(* IEC 61131-3 sources: ai-building-automation/docs/phase0/s3_evidence/dev2/types/generated, 3 files *)

(* ---- PLC_PRG.st ---- *)
PROGRAM PLC_PRG
VAR
    (* Deterministic demo for AHU-01 *)
    StartCommand : BOOL := FALSE;
    StopCommand : BOOL := FALSE;
    FanCommand : BOOL := FALSE;
    FanRunning : BOOL := FALSE;
    FanFault : BOOL := FALSE;
    SupplyTemp : REAL := 21.0;
    Setpoint : REAL := 22.0;
    FanSpeed : REAL := 50.0;
    HeatingValve : REAL := 0.0;
    TestCoil : BOOL := FALSE;
    TestDiscreteInput : BOOL := TRUE;
    TestWordRead : WORD := 16#A55A;
    TestWordWrite : WORD := 16#0000;
    TestInt16Read : INT := -1234;
    TestInt16Write : INT := 0;
    TestUInt16Read : UINT := 1234;
    TestUInt16Write : UINT := 0;
    TestReal32Read : REAL := 21.5;
    TestReal32Write : REAL := 0.0;
    (* Modbus TCP image (16-bit words, mapped to Modbus_TCP_Server I/O) *)
    Mb_Command : WORD; (* HR0 Command: bit0=StartCommand, bit1=StopCommand *)
    Mb_TestInt16Write : WORD; (* HR1 TestInt16Write INT16 WRITE *)
    Mb_TestReal32Write_W0 : WORD; (* HR2 TestReal32Write REAL32 memory word 0 *)
    Mb_TestReal32Write_W1 : WORD; (* HR3 TestReal32Write REAL32 memory word 1 *)
    p_TestReal32Write : POINTER TO ARRAY[0..1] OF WORD;
    Mb_TestUInt16Write : WORD; (* HR4 TestUInt16Write UINT16 WRITE *)
    Mb_Status : WORD; (* IR0 Status: bit0=FanCommand, bit1=FanRunning, bit2=FanFault *)
    Mb_TestInt16Read : WORD; (* IR1 TestInt16Read INT16 READ *)
    Mb_TestReal32Read_W0 : WORD; (* IR2 TestReal32Read REAL32 memory word 0 *)
    Mb_TestReal32Read_W1 : WORD; (* IR3 TestReal32Read REAL32 memory word 1 *)
    p_TestReal32Read : POINTER TO ARRAY[0..1] OF WORD;
    Mb_TestUInt16Read : WORD; (* IR4 TestUInt16Read UINT16 READ *)
END_VAR

(* MODBUS IN: HR0 Command word -> commands *)
StartCommand := Mb_Command.0;
StopCommand := Mb_Command.1;

(* MODBUS IN: HR1 TestInt16Write INT16 *)
TestInt16Write := WORD_TO_INT(Mb_TestInt16Write);

(* MODBUS IN: HR2..HR3 TestReal32Write REAL32 (register words -> REAL memory) *)
p_TestReal32Write := ADR(TestReal32Write);
p_TestReal32Write^[0] := Mb_TestReal32Write_W0;
p_TestReal32Write^[1] := Mb_TestReal32Write_W1;

(* MODBUS IN: HR4 TestUInt16Write UINT16 *)
TestUInt16Write := WORD_TO_UINT(Mb_TestUInt16Write);

(* FAN START *)
IF StartCommand = TRUE AND FanFault = FALSE THEN
    FanCommand := TRUE;
    FanRunning := TRUE;
END_IF;

(* FAN STOP *)
IF StopCommand = TRUE THEN
    FanCommand := FALSE;
    FanRunning := FALSE;
END_IF;

(* FAN FAULT *)
IF FanFault = TRUE THEN
    FanCommand := FALSE;
    FanRunning := FALSE;
END_IF;

(* HEATING - simple demo, not PID *)
IF SupplyTemp < Setpoint THEN
    HeatingValve := 100.0;
ELSE
    HeatingValve := 0.0;
END_IF;

(* MODBUS OUT: status -> IR0 Status word *)
Mb_Status := 0;
Mb_Status.0 := FanCommand;
Mb_Status.1 := FanRunning;
Mb_Status.2 := FanFault;

(* MODBUS OUT: TestInt16Read INT16 -> IR1 *)
Mb_TestInt16Read := INT_TO_WORD(TestInt16Read);

(* MODBUS OUT: TestReal32Read REAL32 (REAL memory -> register words) -> IR2..IR3 *)
p_TestReal32Read := ADR(TestReal32Read);
Mb_TestReal32Read_W0 := p_TestReal32Read^[0];
Mb_TestReal32Read_W1 := p_TestReal32Read^[1];

(* MODBUS OUT: TestUInt16Read UINT16 -> IR4 *)
Mb_TestUInt16Read := UINT_TO_WORD(TestUInt16Read);

(* ---- PLC_PRG_decl.st ---- *)
PROGRAM PLC_PRG
VAR
    (* Deterministic demo for AHU-01 *)
    StartCommand : BOOL := FALSE;
    StopCommand : BOOL := FALSE;
    FanCommand : BOOL := FALSE;
    FanRunning : BOOL := FALSE;
    FanFault : BOOL := FALSE;
    SupplyTemp : REAL := 21.0;
    Setpoint : REAL := 22.0;
    FanSpeed : REAL := 50.0;
    HeatingValve : REAL := 0.0;
    TestCoil : BOOL := FALSE;
    TestDiscreteInput : BOOL := TRUE;
    TestWordRead : WORD := 16#A55A;
    TestWordWrite : WORD := 16#0000;
    TestInt16Read : INT := -1234;
    TestInt16Write : INT := 0;
    TestUInt16Read : UINT := 1234;
    TestUInt16Write : UINT := 0;
    TestReal32Read : REAL := 21.5;
    TestReal32Write : REAL := 0.0;
    (* Modbus TCP image (16-bit words, mapped to Modbus_TCP_Server I/O) *)
    Mb_Command : WORD; (* HR0 Command: bit0=StartCommand, bit1=StopCommand *)
    Mb_TestInt16Write : WORD; (* HR1 TestInt16Write INT16 WRITE *)
    Mb_TestReal32Write_W0 : WORD; (* HR2 TestReal32Write REAL32 memory word 0 *)
    Mb_TestReal32Write_W1 : WORD; (* HR3 TestReal32Write REAL32 memory word 1 *)
    p_TestReal32Write : POINTER TO ARRAY[0..1] OF WORD;
    Mb_TestUInt16Write : WORD; (* HR4 TestUInt16Write UINT16 WRITE *)
    Mb_Status : WORD; (* IR0 Status: bit0=FanCommand, bit1=FanRunning, bit2=FanFault *)
    Mb_TestInt16Read : WORD; (* IR1 TestInt16Read INT16 READ *)
    Mb_TestReal32Read_W0 : WORD; (* IR2 TestReal32Read REAL32 memory word 0 *)
    Mb_TestReal32Read_W1 : WORD; (* IR3 TestReal32Read REAL32 memory word 1 *)
    p_TestReal32Read : POINTER TO ARRAY[0..1] OF WORD;
    Mb_TestUInt16Read : WORD; (* IR4 TestUInt16Read UINT16 READ *)
END_VAR

(* ---- PLC_PRG_impl.st ---- *)
(* MODBUS IN: HR0 Command word -> commands *)
StartCommand := Mb_Command.0;
StopCommand := Mb_Command.1;

(* MODBUS IN: HR1 TestInt16Write INT16 *)
TestInt16Write := WORD_TO_INT(Mb_TestInt16Write);

(* MODBUS IN: HR2..HR3 TestReal32Write REAL32 (register words -> REAL memory) *)
p_TestReal32Write := ADR(TestReal32Write);
p_TestReal32Write^[0] := Mb_TestReal32Write_W0;
p_TestReal32Write^[1] := Mb_TestReal32Write_W1;

(* MODBUS IN: HR4 TestUInt16Write UINT16 *)
TestUInt16Write := WORD_TO_UINT(Mb_TestUInt16Write);

(* FAN START *)
IF StartCommand = TRUE AND FanFault = FALSE THEN
    FanCommand := TRUE;
    FanRunning := TRUE;
END_IF;

(* FAN STOP *)
IF StopCommand = TRUE THEN
    FanCommand := FALSE;
    FanRunning := FALSE;
END_IF;

(* FAN FAULT *)
IF FanFault = TRUE THEN
    FanCommand := FALSE;
    FanRunning := FALSE;
END_IF;

(* HEATING - simple demo, not PID *)
IF SupplyTemp < Setpoint THEN
    HeatingValve := 100.0;
ELSE
    HeatingValve := 0.0;
END_IF;

(* MODBUS OUT: status -> IR0 Status word *)
Mb_Status := 0;
Mb_Status.0 := FanCommand;
Mb_Status.1 := FanRunning;
Mb_Status.2 := FanFault;

(* MODBUS OUT: TestInt16Read INT16 -> IR1 *)
Mb_TestInt16Read := INT_TO_WORD(TestInt16Read);

(* MODBUS OUT: TestReal32Read REAL32 (REAL memory -> register words) -> IR2..IR3 *)
p_TestReal32Read := ADR(TestReal32Read);
Mb_TestReal32Read_W0 := p_TestReal32Read^[0];
Mb_TestReal32Read_W1 := p_TestReal32Read^[1];

(* MODBUS OUT: TestUInt16Read UINT16 -> IR4 *)
Mb_TestUInt16Read := UINT_TO_WORD(TestUInt16Read);
